PROGRAM S1_01_RobPickPart_1
VAR
	HMI_Motion: FB_HMI_Control;
	Motion: FB_Motion2way;

	tMessageOffset: UINT;
	tNumMessagesPerRow: UINT;
	
	
	MyAdvanceInterlock: BOOL;
	MyReturnInterlock: BOOL;
	
	MyAutoAdvanceCondition: BOOL;
	MyAutoReturnCondition: BOOL;
	testword: WORD;
	myAdvancePrompt: BOOL;
	myReturnPrompt: BOOL;
	advancedSensor: BOOL;
	returnedSensor: BOOL;
	AdvanceCoil: BOOL;
	ReturnCoil: BOOL;
	FB_Step_0: FB_Step;
	FB_Step_1: FB_Step;
	FB_Step_2: FB_Step;
	FB_Step_3: FB_Step;
	FB_Step_4: FB_Step;
	FB_Step_5: FB_Step;
	FB_Step_6: FB_Step;
	FB_Step_7: FB_Step;
	tWaitMsgXICAdv: BOOL;
	tWaitMsgXICRet: BOOL;
	FB_GetStateAutoRow_0: FB_GetStateAutoRow;

	robToPickPart: FB_RobotMotion;
	robToHome: FB_RobotMotion;
END_VAR

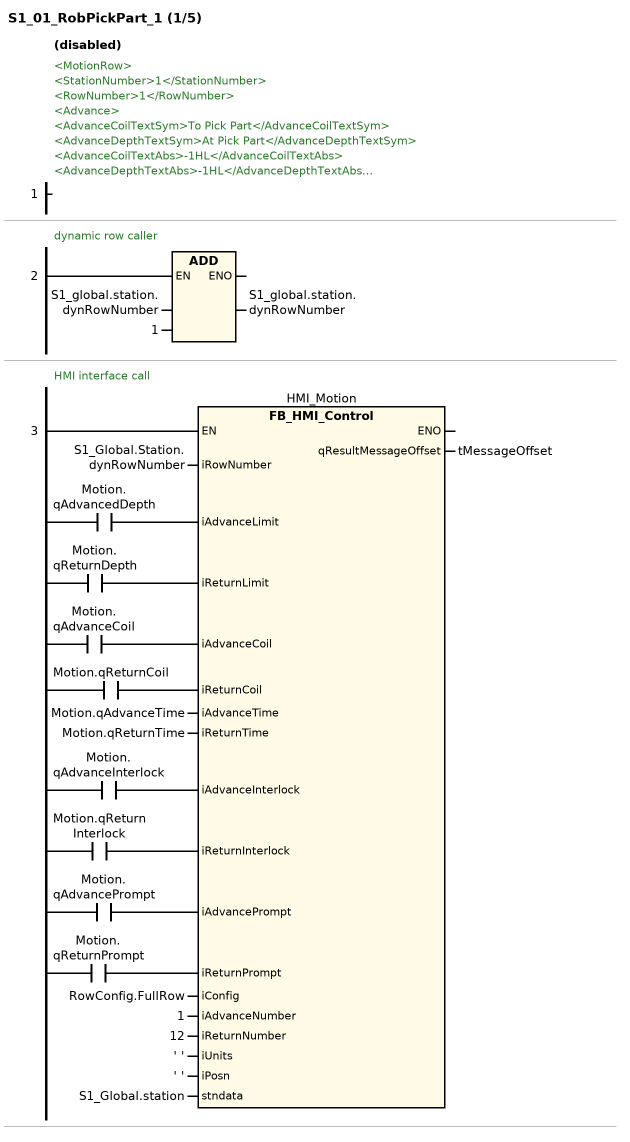
// NETWORK 1 (disabled)
// <MotionRow>
// <StationNumber>1</StationNumber>
// <RowNumber>1</RowNumber>
//   <Advance>
//     <AdvanceCoilTextSym>To Pick Part</AdvanceCoilTextSym>
//     <AdvanceDepthTextSym>At Pick Part</AdvanceDepthTextSym>
//     <AdvanceCoilTextAbs>-1HL</AdvanceCoilTextAbs>
//     <AdvanceDepthTextAbs>-1HL</AdvanceDepthTextAbs>
//     <ManSeq>1</ManSeq>
//   </Advance>
//   <Return>
//     <ReturnCoilTextSym>To Home</ReturnCoilTextSym>
//     <ReturnDepthTextSym>At Home</ReturnDepthTextSym>
//     <ReturnCoilTextAbs>-1HL</ReturnCoilTextAbs>
//     <ReturnDepthTextAbs>-1HL</ReturnDepthTextAbs>
//    <ManSeq>12</ManSeq>
//   </Return>
//   <Motion>
//     <NameSym>Robot</NameSym>
//     <NameAbs>-1HL</NameAbs>
//   </Motion>
// </MotionRow>

// NETWORK 2
// dynamic row caller
S1_global.station.dynRowNumber := S1_global.station.dynRowNumber + 1;

// NETWORK 3
// HMI interface call
HMI_Motion(
    iRowNumber := S1_Global.Station.dynRowNumber,
    iAdvanceLimit := Motion.qAdvancedDepth,
    iReturnLimit := Motion.qReturnDepth,
    iAdvanceCoil := Motion.qAdvanceCoil,
    iReturnCoil := Motion.qReturnCoil,
    iAdvanceTime := Motion.qAdvanceTime,
    iReturnTime := Motion.qReturnTime,
    iAdvanceInterlock := Motion.qAdvanceInterlock,
    iReturnInterlock := Motion.qReturnInterlock,
    iAdvancePrompt := Motion.qAdvancePrompt,
    iReturnPrompt := Motion.qReturnPrompt,
    iConfig := RowConfig.FullRow,
    iAdvanceNumber := 1,
    iReturnNumber := 12,
    iUnits := ' ',
    iPosn := ' ',
    stndata := S1_Global.station,
    qResultMessageOffset => tMessageOffset); // FB_HMI_Control

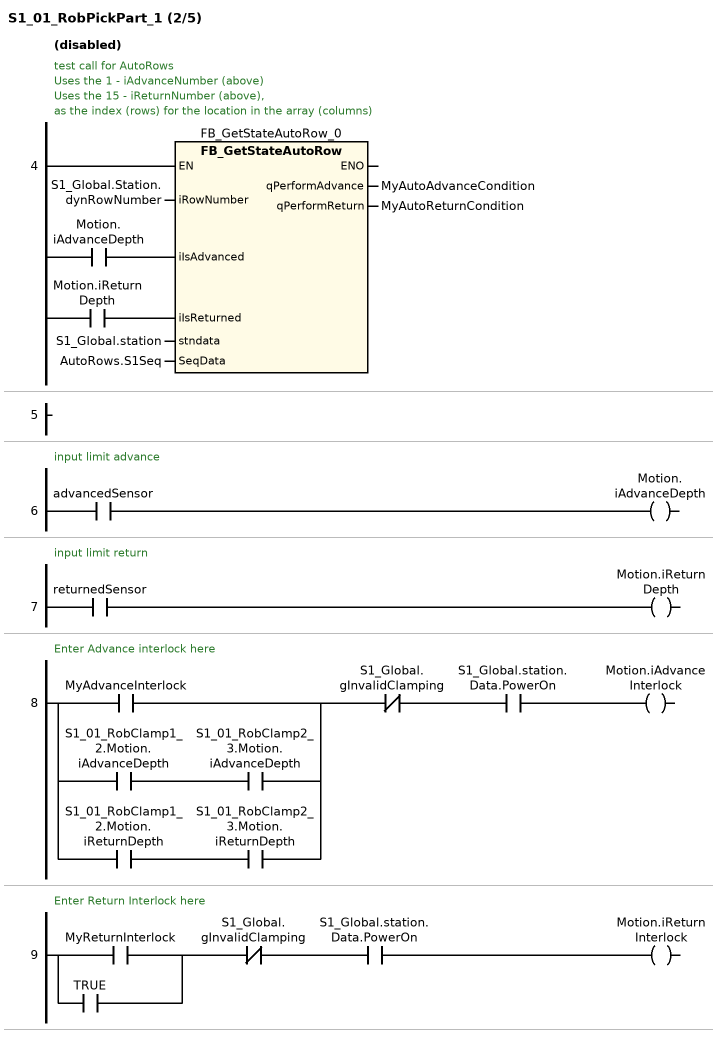
// NETWORK 4 (disabled)
// test call for AutoRows
// Uses the 1 - iAdvanceNumber (above)
// Uses the 15 - iReturnNumber (above),
// as the index (rows) for the location in the array (columns)
// FB_GetStateAutoRow_0(
//     iRowNumber := S1_Global.Station.dynRowNumber,
//     iIsAdvanced := Motion.iAdvanceDepth,
//     iIsReturned := Motion.iReturnDepth,
//     stndata := S1_Global.station,
//     SeqData := AutoRows.S1Seq,
//     qPerformAdvance => MyAutoAdvanceCondition,
//     qPerformReturn => MyAutoReturnCondition); // FB_GetStateAutoRow

// NETWORK 5

// NETWORK 6
// input limit advance
Motion.iAdvanceDepth := advancedSensor;

// NETWORK 7
// input limit return
Motion.iReturnDepth := returnedSensor;

// NETWORK 8
// Enter Advance interlock here
Motion.iAdvanceInterlock := (MyAdvanceInterlock OR S1_01_RobClamp1_2.Motion.iAdvanceDepth AND S1_01_RobClamp2_3.Motion.iAdvanceDepth OR S1_01_RobClamp1_2.Motion.iReturnDepth AND S1_01_RobClamp2_3.Motion.iReturnDepth) AND NOT S1_Global.gInvalidClamping AND S1_Global.station.Data.PowerOn;

// NETWORK 9
// Enter Return Interlock here
Motion.iReturnInterlock := (MyReturnInterlock OR TRUE) AND NOT S1_Global.gInvalidClamping AND S1_Global.station.Data.PowerOn;

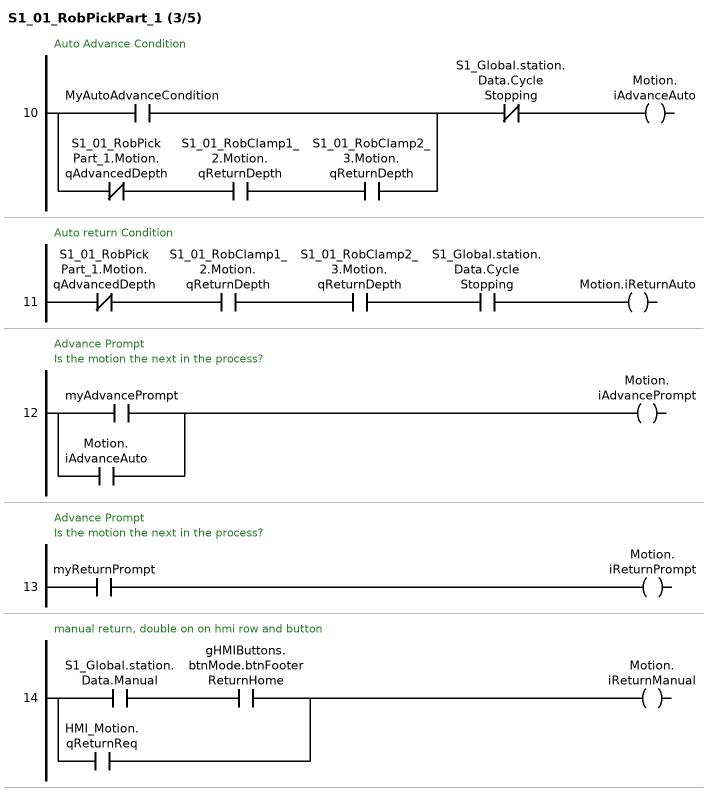
// NETWORK 10
// Auto Advance Condition
Motion.iAdvanceAuto := (MyAutoAdvanceCondition OR NOT S1_01_RobPickPart_1.Motion.qAdvancedDepth AND S1_01_RobClamp1_2.Motion.qReturnDepth AND S1_01_RobClamp2_3.Motion.qReturnDepth) AND NOT S1_Global.station.Data.CycleStopping;

// NETWORK 11
// Auto return Condition
Motion.iReturnAuto := NOT S1_01_RobPickPart_1.Motion.qAdvancedDepth AND S1_01_RobClamp1_2.Motion.qReturnDepth AND S1_01_RobClamp2_3.Motion.qReturnDepth AND S1_Global.station.Data.CycleStopping;

// NETWORK 12
// Advance Prompt
// Is the motion the next in the process?
Motion.iAdvancePrompt := myAdvancePrompt OR Motion.iAdvanceAuto;

// NETWORK 13
// Advance Prompt
// Is the motion the next in the process?
Motion.iReturnPrompt := myReturnPrompt;

// NETWORK 14
// manual return, double on on hmi row and button
Motion.iReturnManual := S1_Global.station.Data.Manual AND gHMIButtons.btnMode.btnFooterReturnHome OR HMI_Motion.qReturnReq;

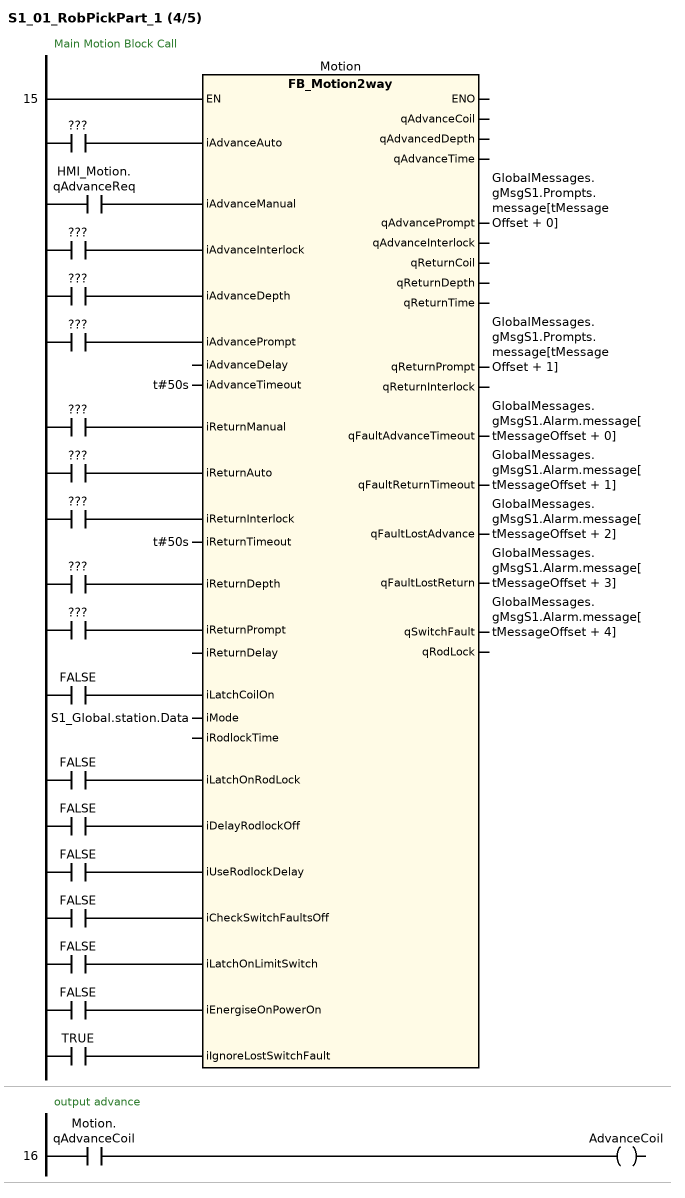
// NETWORK 15
// Main Motion Block Call
Motion(
    iAdvanceManual := HMI_Motion.qAdvanceReq,
    iAdvanceTimeout := t#50s,
    iReturnTimeout := t#50s,
    iLatchCoilOn := FALSE,
    iMode := S1_Global.station.Data,
    iLatchOnRodLock := FALSE,
    iDelayRodlockOff := FALSE,
    iUseRodlockDelay := FALSE,
    iCheckSwitchFaultsOff := FALSE,
    iLatchOnLimitSwitch := FALSE,
    iEnergiseOnPowerOn := FALSE,
    iIgnoreLostSwitchFault := TRUE,
    qAdvancePrompt => GlobalMessages.gMsgS1.Prompts.message[tMessageOffset + 0],
    qReturnPrompt => GlobalMessages.gMsgS1.Prompts.message[tMessageOffset + 1],
    qFaultAdvanceTimeout => GlobalMessages.gMsgS1.Alarm.message[tMessageOffset + 0],
    qFaultReturnTimeout => GlobalMessages.gMsgS1.Alarm.message[tMessageOffset + 1],
    qFaultLostAdvance => GlobalMessages.gMsgS1.Alarm.message[tMessageOffset + 2],
    qFaultLostReturn => GlobalMessages.gMsgS1.Alarm.message[tMessageOffset + 3],
    qSwitchFault => GlobalMessages.gMsgS1.Alarm.message[tMessageOffset + 4]); // FB_Motion2way

// NETWORK 16
// output advance
AdvanceCoil := Motion.qAdvanceCoil;

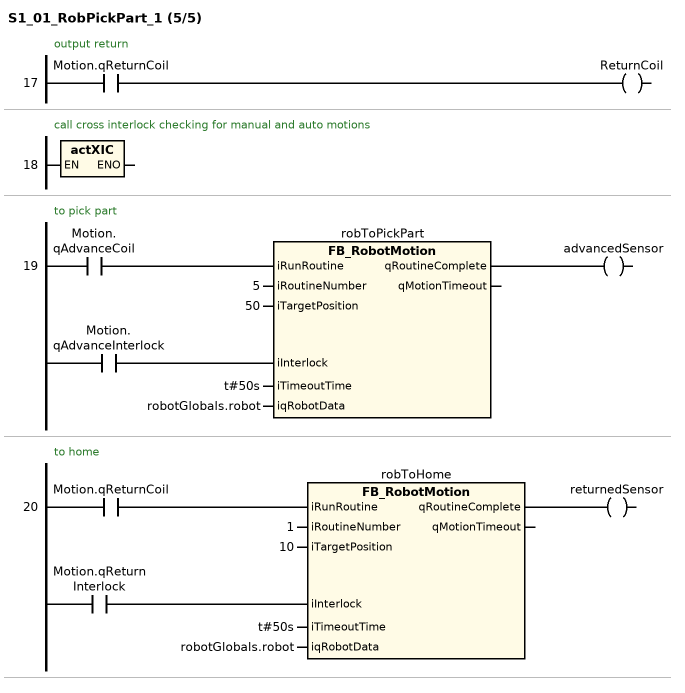
// NETWORK 17
// output return
ReturnCoil := Motion.qReturnCoil;

// NETWORK 18
// call cross interlock checking for manual and auto motions
actXIC();

// NETWORK 19
// to pick part
robToPickPart(
    iRunRoutine := Motion.qAdvanceCoil,
    iRoutineNumber := 5,
    iTargetPosition := 50,
    iInterlock := Motion.qAdvanceInterlock,
    iTimeoutTime := t#50s,
    iqRobotData := robotGlobals.robot); // FB_RobotMotion
advancedSensor := robToPickPart.qRoutineComplete;

// NETWORK 20
// to home
robToHome(
    iRunRoutine := Motion.qReturnCoil,
    iRoutineNumber := 1,
    iTargetPosition := 10,
    iInterlock := Motion.qReturnInterlock,
    iTimeoutTime := t#50s,
    iqRobotData := robotGlobals.robot); // FB_RobotMotion
returnedSensor := robToHome.qRoutineComplete;

ACTION actXIC:
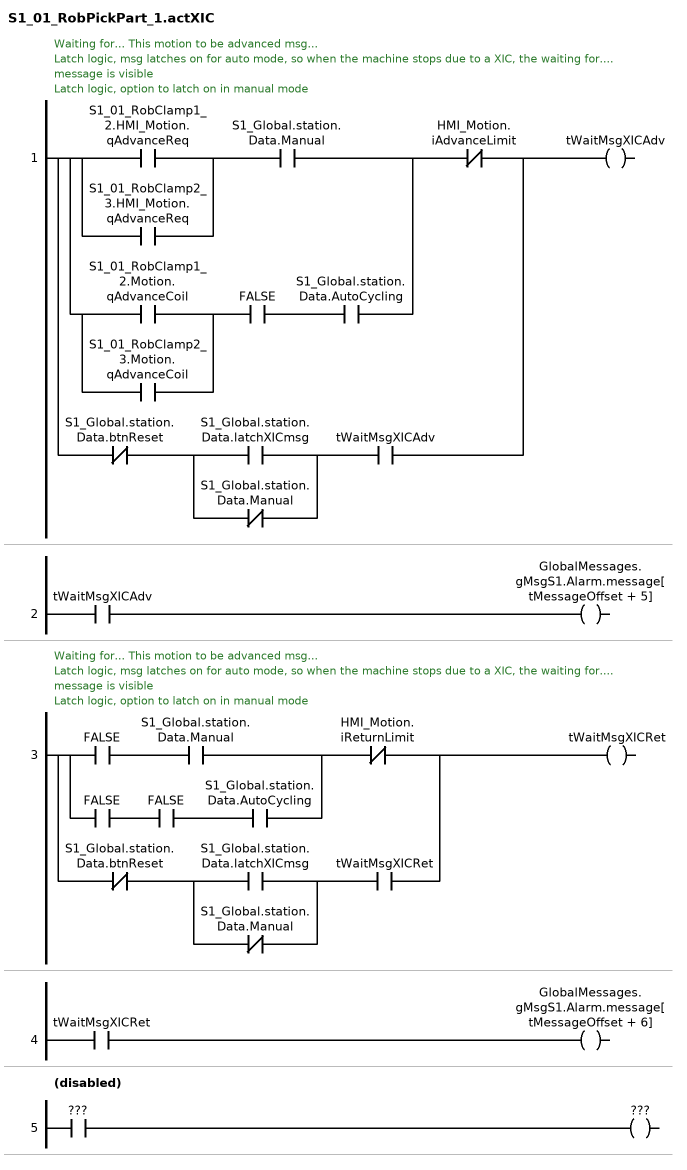
// NETWORK 1
// Waiting for... This motion to be advanced msg...
// Latch logic, msg latches on for auto mode, so when the machine stops due to a XIC, the waiting for.... message is visible
// Latch logic, option to latch on in manual mode
tWaitMsgXICAdv := ((S1_01_RobClamp1_2.HMI_Motion.qAdvanceReq OR S1_01_RobClamp2_3.HMI_Motion.qAdvanceReq) AND S1_Global.station.Data.Manual OR (S1_01_RobClamp1_2.Motion.qAdvanceCoil OR S1_01_RobClamp2_3.Motion.qAdvanceCoil) AND FALSE AND S1_Global.station.Data.AutoCycling) AND NOT HMI_Motion.iAdvanceLimit OR NOT S1_Global.station.Data.btnReset AND (S1_Global.station.Data.latchXICmsg OR NOT S1_Global.station.Data.Manual) AND tWaitMsgXICAdv;

// NETWORK 2
GlobalMessages.gMsgS1.Alarm.message[tMessageOffset + 5] := tWaitMsgXICAdv;

// NETWORK 3
// Waiting for... This motion to be advanced msg...
// Latch logic, msg latches on for auto mode, so when the machine stops due to a XIC, the waiting for.... message is visible
// Latch logic, option to latch on in manual mode
tWaitMsgXICRet := (FALSE AND S1_Global.station.Data.Manual OR FALSE AND FALSE AND S1_Global.station.Data.AutoCycling) AND NOT HMI_Motion.iReturnLimit OR NOT S1_Global.station.Data.btnReset AND (S1_Global.station.Data.latchXICmsg OR NOT S1_Global.station.Data.Manual) AND tWaitMsgXICRet;

// NETWORK 4
GlobalMessages.gMsgS1.Alarm.message[tMessageOffset + 6] := tWaitMsgXICRet;

// NETWORK 5 (disabled)
// ??? := ???;
END_ACTION

END_PROGRAM

(* stored: Version 1.1.0.1, ProductVersion 3.1.4024.11
   POU S1_01_RobPickPart_1: Id {1e53a64d-2400-4f22-b62f-f085377b9b5e}, SpecialFunc None
   Action actXIC: Id {fa76c93a-5256-0755-1a4d-ee773c3fdf8e} *)
